// TIA Portal project "ASSEMBLER_3_0" (V18)

(* hardware
DEVICE "S7-1200-Station_1"  S7-1200 Station
   slot 0: "Baugruppenträger_0"  Rack  V1.0
   slot 1: "PLC_2"  CPU 1212C DC/DC/DC  6ES7 212-1AE40-0XB0  V4.6
*)

// ===== PLC "PLC_2"  CPU 1212C DC/DC/DC =====

VAR_GLOBAL   // PLC tag table "Standard-Variablentabelle"
   "System_Byte" AT %MB10 : Byte;
   "FirstScan" AT %M10.0 : Bool;
   "DiagStatusUpdate" AT %M10.1 : Bool;
   "AlwaysTRUE" AT %M10.2 : Bool;
   "AlwaysFALSE" AT %M10.3 : Bool;
   "Clock_Byte" AT %MB20 : Byte;
   "Clock_10Hz" AT %M20.0 : Bool;
   "Clock_5Hz" AT %M20.1 : Bool;
   "Clock_2.5Hz" AT %M20.2 : Bool;
   "Clock_2Hz" AT %M20.3 : Bool;
   "Clock_1.25Hz" AT %M20.4 : Bool;
   "Clock_1Hz" AT %M20.5 : Bool;
   "Clock_0.625Hz" AT %M20.6 : Bool;
   "Clock_0.5Hz" AT %M20.7 : Bool;
   "PART_LEAVING_FE_MEM" AT %M0.2 : Bool;
   "COUNTER_SENSOR_FE_MEM" AT %M0.3 : Bool;
END_VAR

VAR_GLOBAL   // PLC tag table "Tag table from XML_1"
   "LID_AT_PLACE" AT %I0.1 : Bool;
   "BASE_AT_PLACE" AT %I0.2 : Bool;
   "PART_LEAVING" AT %I0.3 : Bool;
   "START_BUTTON" AT %I0.4 : Bool;
   "RESET_BUTTON" AT %I0.5 : Bool;
   "STOP_BUTTON" AT %I0.6 : Bool;
   "EMERGENCY_STOP_BUTTON" AT %I0.7 : Bool;
   "AUTO_SELECTOR" AT %I1.0 : Bool;
   "FACTORY I/O (Running)" AT %I1.1 : Bool;
   "LIDS_CONVEYOR_1" AT %Q0.0 : Bool;
   "STOP_BLADE_1" AT %Q0.1 : Bool;
   "LIDS_CONVEYOR_2" AT %Q0.2 : Bool;
   "BASES_CONVEYOR_1" AT %Q0.3 : Bool;
   "STOP_BLADE_2" AT %Q0.4 : Bool;
   "BASES_CONVEYOR_2" AT %Q0.5 : Bool;
   "GRAB" AT %Q0.6 : Bool;
   "GREEN_LIGHT" AT %Q0.7 : Bool;
   "EMERGENCY_LIGHT" AT %Q1.0 : Bool;
   "RED_LIGHT" AT %Q1.1 : Bool;
   "X" AT %ID30 : Real;
   "Z" AT %ID34 : Real;
   "SET_X" AT %QD30 : Real;
   "SET_Z" AT %QD34 : Real;
   "COUNTER" AT %QD38 : DInt;
   "VAL_BUTTON" AT %I1.4 : Bool;
   "MANUAL_SELECTOR" AT %I1.3 : Bool;
   "ITEM_DETECTED" AT %I0.0 : Bool;
   "STOP_REQUEST" AT %M0.0 : Bool;
   "IN_PRODUCTION" AT %M0.1 : Bool;
   "YELLOW_LIGHT" AT %Q1.2 : Bool;
   "COUNT_SENSOR" AT %I1.2 : Bool;
END_VAR

DATA_BLOCK "DB"   // DB1
{ S7_Optimized_Access := 'TRUE' }
VERSION : 0.1
   VAR
      MODE_REPOS : Bool;
      MODE_MANUEL : Bool;
      MODE_AUTO : Bool;
      MODE_ARU : Bool;
   END_VAR
BEGIN
END_DATA_BLOCK

DATA_BLOCK "FB_AUTO_DB"   // DB5
{ S7_Optimized_Access := 'TRUE' }
VERSION : 0.1
// stored: InstanceOfName FB_AUTO
"FB_AUTO"
BEGIN
END_DATA_BLOCK

DATA_BLOCK "FB_MAN_DB"   // DB6
{ S7_Optimized_Access := 'TRUE' }
VERSION : 0.1
// stored: InstanceOfName FB_MAN
"FB_MAN"
BEGIN
END_DATA_BLOCK

// folder: System blocks/Program resources

DATA_BLOCK "IEC_Counter_0_DB"   // DB2
{ S7_Optimized_Access := 'TRUE' }
AUTHOR : Simatic
FAMILY : IEC
NAME : CNTR
VERSION : 1.0
// stored: InstanceOfName IEC_COUNTER
"IEC_COUNTER"
BEGIN
END_DATA_BLOCK

DATA_BLOCK "IEC_Timer_0_DB_2"   // DB3
{ S7_Optimized_Access := 'TRUE' }
AUTHOR : Simatic
FAMILY : IEC
NAME : IEC_TMR
VERSION : 1.0
// stored: InstanceOfName IEC_TIMER
"IEC_TIMER"
BEGIN
END_DATA_BLOCK

DATA_BLOCK "IEC_Timer_0_DB"   // DB4
{ S7_Optimized_Access := 'TRUE' }
AUTHOR : Simatic
FAMILY : IEC
NAME : IEC_TMR
VERSION : 1.0
// stored: InstanceOfName IEC_TIMER
"IEC_TIMER"
BEGIN
END_DATA_BLOCK

// folder: (top level)

FUNCTION_BLOCK "FB_AUTO"   // FB1, LAD
{ S7_Optimized_Access := 'TRUE' }
VERSION : 0.1
   VAR_INPUT
      part_leaving : Bool;
      Item_detected : Bool;
      lid_at_place : Bool;
      base_at_place : Bool;
      start_button : Bool;
   END_VAR
   VAR_OUTPUT
      lids_conveyor_1 : Bool;
      lids_conveyor_2 : Bool;
      stop_blade_1 : Bool;
      bases_conveyor_1 : Bool;
      bases_coveyor_2 : Bool;
      stop_blade_2 : Bool;
      set_x : Real;
      set_z : Real;
   END_VAR
   VAR_IN_OUT
      grab : Bool;
      in_production : Bool;
   END_VAR
   VAR
      brake : Bool;
      assembled : Bool;
      bases_stop_blade_timer : Bool;
      SR_1 : Bool;
      SR_2 : Bool;
      SR_3 : Bool;
      grab_negative : Bool;
      falling_edge_1 : Bool;
      falling_edge_2 : Bool;
   END_VAR
   VAR_TEMP   // added for the SCL form of the ladder/FBD networks
      _w1 : Bool;
      _w2 : Bool;
   END_VAR
BEGIN

REGION Network 1
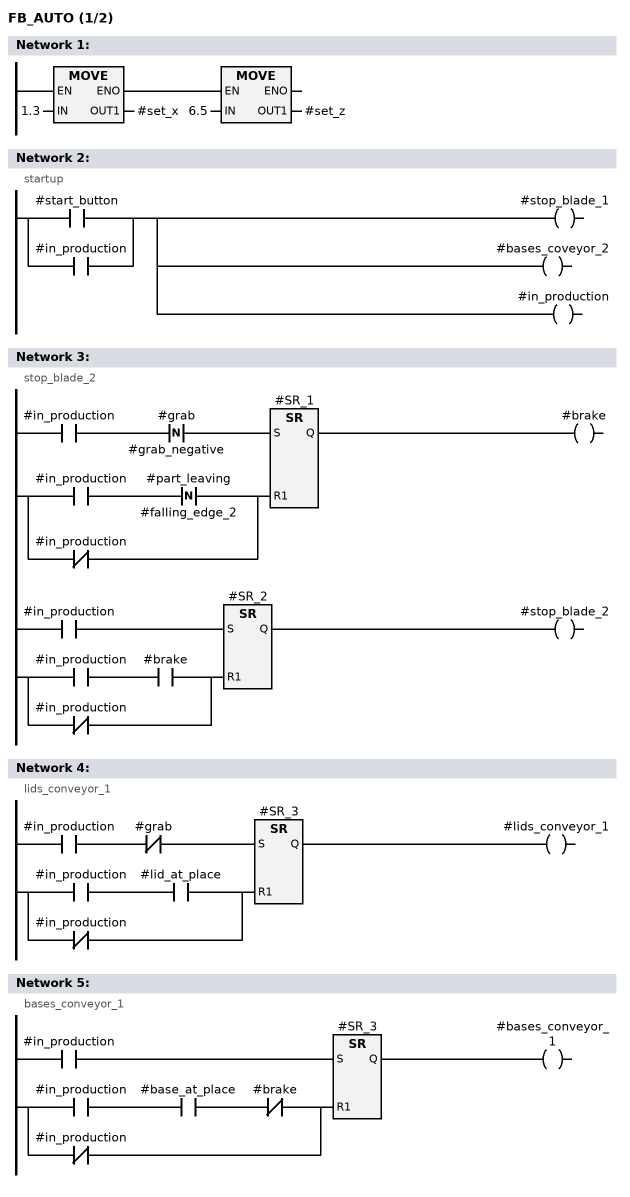
   RUNG wire#powerrail
      Move(in := 1.3, out1 => #set_x)
      Move(in := 6.5, out1 => #set_z)
   END_RUNG
   // the same network as SCL:
   #set_x := 1.3;
   #set_z := 6.5;
END_REGION

REGION Network 2
   // startup
   RUNG wire#powerrail
      Contact( #start_button )
      wire#w1
      Coil( #stop_blade_1 )
   END_RUNG
   RUNG wire#powerrail
      Contact( #in_production )
   END_RUNG wire#w1
   RUNG wire#w1
      Coil( #bases_coveyor_2 )
   END_RUNG
   RUNG wire#w1
      Coil( #in_production )
   END_RUNG
   // the same network as SCL:
   #stop_blade_1 := #start_button OR #in_production;
   #bases_coveyor_2 := #stop_blade_1;
   #in_production := #stop_blade_1;
END_REGION

REGION Network 3
   // stop_blade_2
   RUNG wire#powerrail
      Contact( #in_production )
      N_Contact(operand := #grab, bit := #grab_negative)
      S_SR(operand := #SR_1, r1 := wire#w1)
      Coil( #brake )
   END_RUNG
   RUNG wire#powerrail
      Contact( #in_production )
      N_Contact(operand := #part_leaving, bit := #falling_edge_2)
   END_RUNG wire#w1
   RUNG wire#powerrail
      I_Contact( #in_production )
   END_RUNG wire#w1
   RUNG wire#powerrail
      Contact( #in_production )
      S_SR(operand := #SR_2, r1 := wire#w2)
      Coil( #stop_blade_2 )
   END_RUNG
   RUNG wire#powerrail
      Contact( #in_production )
      Contact( #brake )
   END_RUNG wire#w2
   RUNG wire#powerrail
      I_Contact( #in_production )
   END_RUNG wire#w2
   // the same network as SCL:
   #_w1 := #in_production AND NOT #grab AND #grab_negative;   // falling edge of #grab
   #grab_negative := #grab;
   #_w2 := #in_production AND NOT #part_leaving AND #falling_edge_2;   // falling edge of #part_leaving
   #falling_edge_2 := #part_leaving;
   IF #_w1 THEN
       #SR_1 := TRUE;   // SR flip-flop
   END_IF;
   IF #_w2 OR NOT #in_production THEN #SR_1 := FALSE; END_IF;
   #brake := #SR_1;
   IF #in_production THEN
       #SR_2 := TRUE;   // SR flip-flop
   END_IF;
   IF (#in_production AND #brake) OR NOT #in_production THEN #SR_2 := FALSE; END_IF;
   #stop_blade_2 := #SR_2;
END_REGION

REGION Network 4
   // lids_conveyor_1
   RUNG wire#powerrail
      Contact( #in_production )
      I_Contact( #grab )
      S_SR(operand := #SR_3, r1 := wire#w1)
      Coil( #lids_conveyor_1 )
   END_RUNG
   RUNG wire#powerrail
      Contact( #in_production )
      Contact( #lid_at_place )
   END_RUNG wire#w1
   RUNG wire#powerrail
      I_Contact( #in_production )
   END_RUNG wire#w1
   // the same network as SCL:
   IF #in_production AND NOT #grab THEN
       #SR_3 := TRUE;   // SR flip-flop
   END_IF;
   IF (#in_production AND #lid_at_place) OR NOT #in_production THEN #SR_3 := FALSE; END_IF;
   #lids_conveyor_1 := #SR_3;
END_REGION

REGION Network 5
   // bases_conveyor_1
   RUNG wire#powerrail
      Contact( #in_production )
      S_SR(operand := #SR_3, r1 := wire#w1)
      Coil( #bases_conveyor_1 )
   END_RUNG
   RUNG wire#powerrail
      Contact( #in_production )
      Contact( #base_at_place )
      I_Contact( #brake )
   END_RUNG wire#w1
   RUNG wire#powerrail
      I_Contact( #in_production )
   END_RUNG wire#w1
   // the same network as SCL:
   IF #in_production THEN
       #SR_3 := TRUE;   // SR flip-flop
   END_IF;
   IF (#in_production AND #base_at_place AND NOT #brake) OR NOT #in_production THEN #SR_3 := FALSE; END_IF;
   #bases_conveyor_1 := #SR_3;
END_REGION

REGION Network 6
   // control_de_bras_robotique
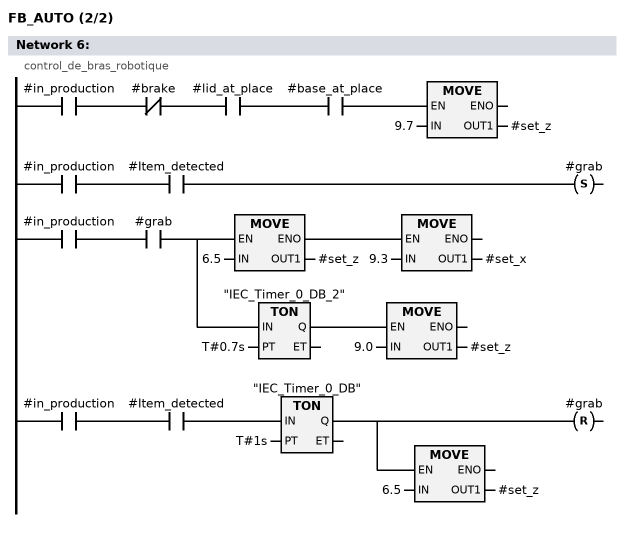
   IF #in_production AND NOT #brake AND #lid_at_place AND #base_at_place THEN #set_z := 9.7; END_IF;
   IF #in_production AND #Item_detected THEN #grab := TRUE; END_IF;
   #_w1 := #in_production AND #grab;
   IF #_w1 THEN
       #set_z := 6.5;
       #set_x := 9.3;
   END_IF;
   "IEC_Timer_0_DB_2".TON(IN := #_w1, PT := T#0.7s);
   IF "IEC_Timer_0_DB_2".Q THEN #set_z := 9.0; END_IF;
   "IEC_Timer_0_DB".TON(IN := #in_production AND #Item_detected, PT := T#1s);
   IF "IEC_Timer_0_DB".Q THEN
       #grab := FALSE;
       #set_z := 6.5;
   END_IF;
END_REGION
END_FUNCTION_BLOCK

FUNCTION_BLOCK "FB_MAN"   // FB2, LAD
{ S7_Optimized_Access := 'TRUE' }
VERSION : 0.1
   VAR_INPUT
      part_leaving : Bool;
      Item_detected : Bool;
      lid_at_place : Bool;
      base_at_place : Bool;
      start_button : Bool;
   END_VAR
   VAR_OUTPUT
      lids_conveyor_1 : Bool;
      lids_conveyor_2 : Bool;
      stop_blade_1 : Bool;
      bases_conveyor_1 : Bool;
      bases_coveyor_2 : Bool;
      stop_blade_2 : Bool;
      set_x : Real;
      set_z : Real;
   END_VAR
   VAR_IN_OUT
      grab : Bool;
      in_production : Bool;
   END_VAR
   VAR
      brake : Bool;
      assembled : Bool;
      bases_stop_blade_timer : Bool;
      SR_1 : Bool;
      SR_2 : Bool;
      SR_3 : Bool;
      grab_negative : Bool;
      falling_edge_1 : Bool;
      falling_edge_2 : Bool;
   END_VAR
   VAR_TEMP   // added for the SCL form of the ladder/FBD networks
      _w1 : Bool;
      _w2 : Bool;
   END_VAR
BEGIN

REGION Network 1
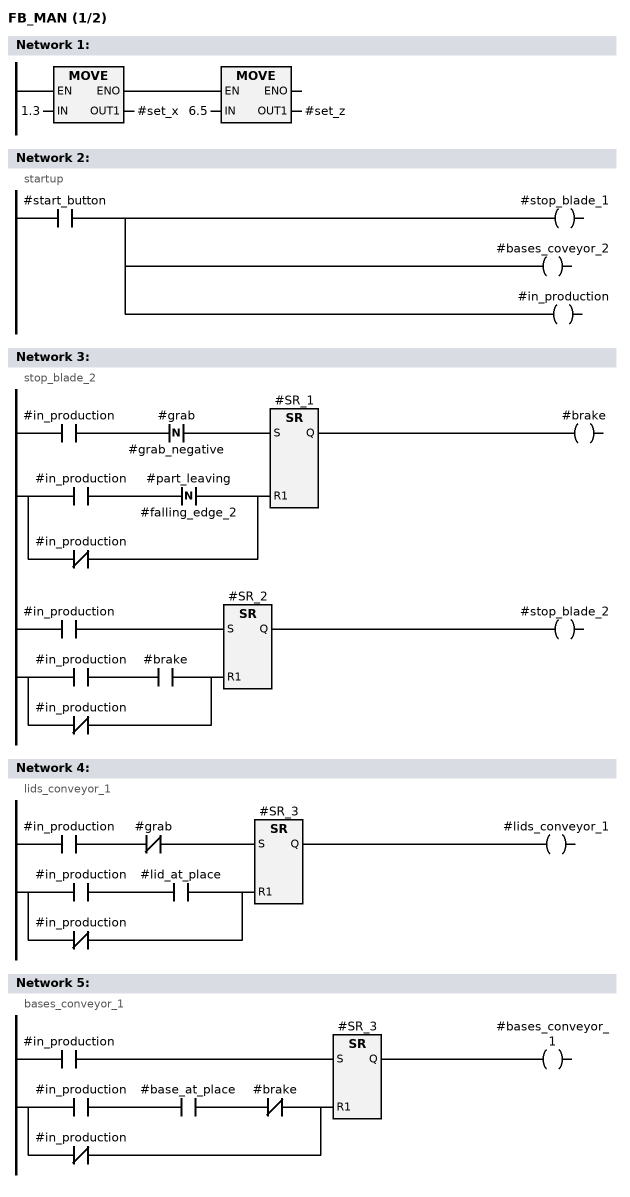
   RUNG wire#powerrail
      Move(in := 1.3, out1 => #set_x)
      Move(in := 6.5, out1 => #set_z)
   END_RUNG
   // the same network as SCL:
   #set_x := 1.3;
   #set_z := 6.5;
END_REGION

REGION Network 2
   // startup
   RUNG wire#powerrail
      Contact( #start_button )
      wire#w1
      Coil( #stop_blade_1 )
   END_RUNG
   RUNG wire#w1
      Coil( #bases_coveyor_2 )
   END_RUNG
   RUNG wire#w1
      Coil( #in_production )
   END_RUNG
   // the same network as SCL:
   #stop_blade_1 := #start_button;
   #bases_coveyor_2 := #start_button;
   #in_production := #start_button;
END_REGION

REGION Network 3
   // stop_blade_2
   RUNG wire#powerrail
      Contact( #in_production )
      N_Contact(operand := #grab, bit := #grab_negative)
      S_SR(operand := #SR_1, r1 := wire#w1)
      Coil( #brake )
   END_RUNG
   RUNG wire#powerrail
      Contact( #in_production )
      N_Contact(operand := #part_leaving, bit := #falling_edge_2)
   END_RUNG wire#w1
   RUNG wire#powerrail
      I_Contact( #in_production )
   END_RUNG wire#w1
   RUNG wire#powerrail
      Contact( #in_production )
      S_SR(operand := #SR_2, r1 := wire#w2)
      Coil( #stop_blade_2 )
   END_RUNG
   RUNG wire#powerrail
      Contact( #in_production )
      Contact( #brake )
   END_RUNG wire#w2
   RUNG wire#powerrail
      I_Contact( #in_production )
   END_RUNG wire#w2
   // the same network as SCL:
   #_w1 := #in_production AND NOT #grab AND #grab_negative;   // falling edge of #grab
   #grab_negative := #grab;
   #_w2 := #in_production AND NOT #part_leaving AND #falling_edge_2;   // falling edge of #part_leaving
   #falling_edge_2 := #part_leaving;
   IF #_w1 THEN
       #SR_1 := TRUE;   // SR flip-flop
   END_IF;
   IF #_w2 OR NOT #in_production THEN #SR_1 := FALSE; END_IF;
   #brake := #SR_1;
   IF #in_production THEN
       #SR_2 := TRUE;   // SR flip-flop
   END_IF;
   IF (#in_production AND #brake) OR NOT #in_production THEN #SR_2 := FALSE; END_IF;
   #stop_blade_2 := #SR_2;
END_REGION

REGION Network 4
   // lids_conveyor_1
   RUNG wire#powerrail
      Contact( #in_production )
      I_Contact( #grab )
      S_SR(operand := #SR_3, r1 := wire#w1)
      Coil( #lids_conveyor_1 )
   END_RUNG
   RUNG wire#powerrail
      Contact( #in_production )
      Contact( #lid_at_place )
   END_RUNG wire#w1
   RUNG wire#powerrail
      I_Contact( #in_production )
   END_RUNG wire#w1
   // the same network as SCL:
   IF #in_production AND NOT #grab THEN
       #SR_3 := TRUE;   // SR flip-flop
   END_IF;
   IF (#in_production AND #lid_at_place) OR NOT #in_production THEN #SR_3 := FALSE; END_IF;
   #lids_conveyor_1 := #SR_3;
END_REGION

REGION Network 5
   // bases_conveyor_1
   RUNG wire#powerrail
      Contact( #in_production )
      S_SR(operand := #SR_3, r1 := wire#w1)
      Coil( #bases_conveyor_1 )
   END_RUNG
   RUNG wire#powerrail
      Contact( #in_production )
      Contact( #base_at_place )
      I_Contact( #brake )
   END_RUNG wire#w1
   RUNG wire#powerrail
      I_Contact( #in_production )
   END_RUNG wire#w1
   // the same network as SCL:
   IF #in_production THEN
       #SR_3 := TRUE;   // SR flip-flop
   END_IF;
   IF (#in_production AND #base_at_place AND NOT #brake) OR NOT #in_production THEN #SR_3 := FALSE; END_IF;
   #bases_conveyor_1 := #SR_3;
END_REGION

REGION Network 6
   // control_de_bras_robotique
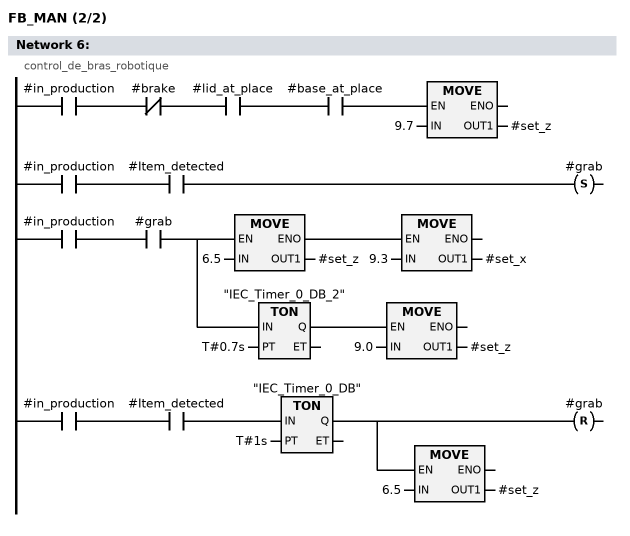
   IF #in_production AND NOT #brake AND #lid_at_place AND #base_at_place THEN #set_z := 9.7; END_IF;
   IF #in_production AND #Item_detected THEN #grab := TRUE; END_IF;
   #_w1 := #in_production AND #grab;
   IF #_w1 THEN
       #set_z := 6.5;
       #set_x := 9.3;
   END_IF;
   "IEC_Timer_0_DB_2".TON(IN := #_w1, PT := T#0.7s);
   IF "IEC_Timer_0_DB_2".Q THEN #set_z := 9.0; END_IF;
   "IEC_Timer_0_DB".TON(IN := #in_production AND #Item_detected, PT := T#1s);
   IF "IEC_Timer_0_DB".Q THEN
       #grab := FALSE;
       #set_z := 6.5;
   END_IF;
END_REGION
END_FUNCTION_BLOCK

FUNCTION "FC_ARU_REPOS" : Void   // FC2, LAD
{ S7_Optimized_Access := 'TRUE' }
VERSION : 0.1
   VAR_OUTPUT
      lids_conveyor_1 : Bool;
      lids_conveyor_2 : Bool;
      stop_blade_1 : Bool;
      bases_conveyor_1 : Bool;
      bases_coveyor_2 : Bool;
      stop_blade_2 : Bool;
   END_VAR
   VAR_IN_OUT
      grab : Bool;
   END_VAR
BEGIN

REGION Network 1
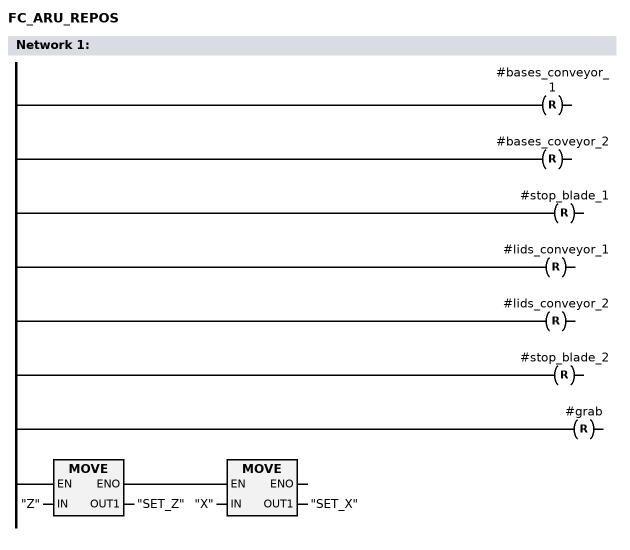
   RUNG wire#powerrail
      R_Coil( #bases_conveyor_1 )
   END_RUNG
   RUNG wire#powerrail
      R_Coil( #bases_coveyor_2 )
   END_RUNG
   RUNG wire#powerrail
      R_Coil( #stop_blade_1 )
   END_RUNG
   RUNG wire#powerrail
      R_Coil( #lids_conveyor_1 )
   END_RUNG
   RUNG wire#powerrail
      R_Coil( #lids_conveyor_2 )
   END_RUNG
   RUNG wire#powerrail
      R_Coil( #stop_blade_2 )
   END_RUNG
   RUNG wire#powerrail
      R_Coil( #grab )
   END_RUNG
   RUNG wire#powerrail
      Move(in := "Z", out1 => "SET_Z")
      Move(in := "X", out1 => "SET_X")
   END_RUNG
   // the same network as SCL:
   #bases_conveyor_1 := FALSE;
   #bases_coveyor_2 := FALSE;
   #stop_blade_1 := FALSE;
   #lids_conveyor_1 := FALSE;
   #lids_conveyor_2 := FALSE;
   #stop_blade_2 := FALSE;
   #grab := FALSE;
   "SET_Z" := "Z";
   "SET_X" := "X";
END_REGION
END_FUNCTION

FUNCTION "FC_MODES_GEST" : Void   // FC5, LAD
{ S7_Optimized_Access := 'TRUE' }
VERSION : 0.1
   VAR_INPUT
      stop_button : Bool;
      auto_selector : Bool;
      val_button : Bool;
      manual_selector : Bool;
      emergency_stop_button : Bool;
      part_leaving : Bool;
   END_VAR
   VAR_OUTPUT
      green_light : Bool;
      yellow_light : Bool;
      red_light : Bool;
      emergency_light : Bool;
   END_VAR
   VAR_IN_OUT
      mode_man : Bool;
      mode_repos : Bool;
      mode_auto : Bool;
      mode_aru : Bool;
      in_production : Bool;
   END_VAR
   VAR_TEMP   // added for the SCL form of the ladder/FBD networks
      _w1 : Bool;
      _w2 : Bool;
   END_VAR
BEGIN

REGION Network 1
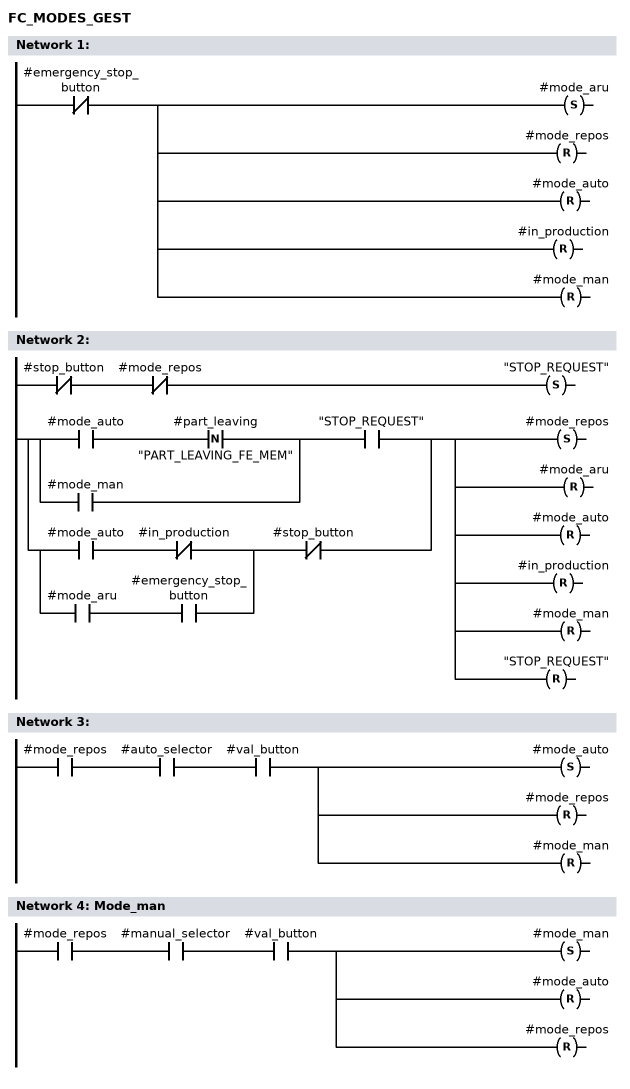
   RUNG wire#powerrail
      I_Contact( #emergency_stop_button )
      wire#w1
      S_Coil( #mode_aru )
   END_RUNG
   RUNG wire#w1
      R_Coil( #mode_repos )
   END_RUNG
   RUNG wire#w1
      R_Coil( #mode_auto )
   END_RUNG
   RUNG wire#w1
      R_Coil( #in_production )
   END_RUNG
   RUNG wire#w1
      R_Coil( #mode_man )
   END_RUNG
   // the same network as SCL:
   IF NOT #emergency_stop_button THEN
       #mode_aru := TRUE;
       #mode_repos := FALSE;
       #mode_auto := FALSE;
       #in_production := FALSE;
       #mode_man := FALSE;
   END_IF;
END_REGION

REGION Network 2
   RUNG wire#powerrail
      I_Contact( #stop_button )
      I_Contact( #mode_repos )
      S_Coil( "STOP_REQUEST" )
   END_RUNG
   RUNG wire#powerrail
      Contact( #mode_auto )
      N_Contact(operand := #part_leaving, bit := "PART_LEAVING_FE_MEM")
      wire#w1
      Contact( "STOP_REQUEST" )
      wire#w2
      S_Coil( #mode_repos )
   END_RUNG
   RUNG wire#powerrail
      Contact( #mode_man )
   END_RUNG wire#w1
   RUNG wire#powerrail
      Contact( #mode_auto )
      I_Contact( #in_production )
      wire#w3
      I_Contact( #stop_button )
   END_RUNG wire#w2
   RUNG wire#powerrail
      Contact( #mode_aru )
      Contact( #emergency_stop_button )
   END_RUNG wire#w3
   RUNG wire#w2
      R_Coil( #mode_aru )
   END_RUNG
   RUNG wire#w2
      R_Coil( #mode_auto )
   END_RUNG
   RUNG wire#w2
      R_Coil( #in_production )
   END_RUNG
   RUNG wire#w2
      R_Coil( #mode_man )
   END_RUNG
   RUNG wire#w2
      R_Coil( "STOP_REQUEST" )
   END_RUNG
   // the same network as SCL:
   IF NOT #stop_button AND NOT #mode_repos THEN "STOP_REQUEST" := TRUE; END_IF;
   #_w1 := #mode_auto AND NOT #part_leaving AND "PART_LEAVING_FE_MEM";   // falling edge of #part_leaving
   "PART_LEAVING_FE_MEM" := #part_leaving;
   IF ((#_w1 OR #mode_man) AND "STOP_REQUEST") OR (((#mode_auto AND NOT #in_production) OR (#mode_aru AND #emergency_stop_button)) AND NOT #stop_button) THEN
       #mode_repos := TRUE;
   END_IF;
   #_w2 := ((#_w1 OR #mode_man) AND "STOP_REQUEST") OR (((#mode_auto AND NOT #in_production) OR (#mode_aru AND #emergency_stop_button)) AND NOT #stop_button);
   IF #_w2 THEN
       #mode_aru := FALSE;
       #mode_auto := FALSE;
       #in_production := FALSE;
       #mode_man := FALSE;
       "STOP_REQUEST" := FALSE;
   END_IF;
END_REGION

REGION Network 3
   RUNG wire#powerrail
      Contact( #mode_repos )
      Contact( #auto_selector )
      Contact( #val_button )
      wire#w1
      S_Coil( #mode_auto )
   END_RUNG
   RUNG wire#w1
      R_Coil( #mode_repos )
   END_RUNG
   RUNG wire#w1
      R_Coil( #mode_man )
   END_RUNG
   // the same network as SCL:
   IF #mode_repos AND #auto_selector AND #val_button THEN #mode_auto := TRUE; END_IF;
   #_w1 := #mode_repos AND #auto_selector AND #val_button;
   IF #_w1 THEN
       #mode_repos := FALSE;
       #mode_man := FALSE;
   END_IF;
END_REGION

REGION Network 4: Mode_man
   RUNG wire#powerrail
      Contact( #mode_repos )
      Contact( #manual_selector )
      Contact( #val_button )
      wire#w1
      S_Coil( #mode_man )
   END_RUNG
   RUNG wire#w1
      R_Coil( #mode_auto )
   END_RUNG
   RUNG wire#w1
      R_Coil( #mode_repos )
   END_RUNG
   // the same network as SCL:
   IF #mode_repos AND #manual_selector AND #val_button THEN
       #mode_man := TRUE;
       #mode_auto := FALSE;
       #mode_repos := FALSE;
   END_IF;
END_REGION
END_FUNCTION

FUNCTION "FC_VOY_GEST" : Void   // FC6, LAD
{ S7_Optimized_Access := 'TRUE' }
VERSION : 0.1
   VAR_OUTPUT
      green_light : Bool;
      yellow_light : Bool;
      red_light : Bool;
      emergency_light : Bool;
   END_VAR
   VAR_IN_OUT
      mode_man : Bool;
      mode_repos : Bool;
      mode_auto : Bool;
      mode_aru : Bool;
      in_production : Bool;
   END_VAR
BEGIN

REGION Network 1
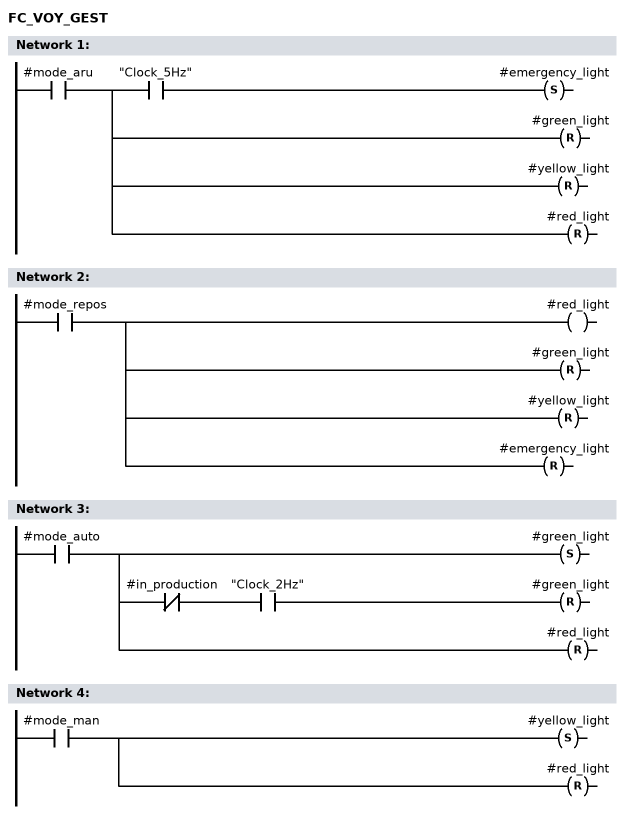
   RUNG wire#powerrail
      Contact( #mode_aru )
      wire#w1
      Contact( "Clock_5Hz" )
      S_Coil( #emergency_light )
   END_RUNG
   RUNG wire#w1
      R_Coil( #green_light )
   END_RUNG
   RUNG wire#w1
      R_Coil( #yellow_light )
   END_RUNG
   RUNG wire#w1
      R_Coil( #red_light )
   END_RUNG
   // the same network as SCL:
   IF #mode_aru AND "Clock_5Hz" THEN #emergency_light := TRUE; END_IF;
   IF #mode_aru THEN
       #green_light := FALSE;
       #yellow_light := FALSE;
       #red_light := FALSE;
   END_IF;
END_REGION

REGION Network 2
   RUNG wire#powerrail
      Contact( #mode_repos )
      wire#w1
      Coil( #red_light )
   END_RUNG
   RUNG wire#w1
      R_Coil( #green_light )
   END_RUNG
   RUNG wire#w1
      R_Coil( #yellow_light )
   END_RUNG
   RUNG wire#w1
      R_Coil( #emergency_light )
   END_RUNG
   // the same network as SCL:
   #red_light := #mode_repos;
   IF #mode_repos THEN
       #green_light := FALSE;
       #yellow_light := FALSE;
       #emergency_light := FALSE;
   END_IF;
END_REGION

REGION Network 3
   RUNG wire#powerrail
      Contact( #mode_auto )
      wire#w1
      S_Coil( #green_light )
   END_RUNG
   RUNG wire#w1
      I_Contact( #in_production )
      Contact( "Clock_2Hz" )
      R_Coil( #green_light )
   END_RUNG
   RUNG wire#w1
      R_Coil( #red_light )
   END_RUNG
   // the same network as SCL:
   IF #mode_auto THEN #green_light := TRUE; END_IF;
   IF #mode_auto AND NOT #in_production AND "Clock_2Hz" THEN #green_light := FALSE; END_IF;
   IF #mode_auto THEN #red_light := FALSE; END_IF;
END_REGION

REGION Network 4
   RUNG wire#powerrail
      Contact( #mode_man )
      wire#w1
      S_Coil( #yellow_light )
   END_RUNG
   RUNG wire#w1
      R_Coil( #red_light )
   END_RUNG
   // the same network as SCL:
   IF #mode_man THEN
       #yellow_light := TRUE;
       #red_light := FALSE;
   END_IF;
END_REGION

REGION Network 6: Mode_man
END_REGION
END_FUNCTION

FUNCTION "Factory_IO" : Void   // FC9000, SCL
{ S7_Optimized_Access := 'TRUE' }
VERSION : 0.1
   VAR_TEMP
      rdTimeReturn : Int;
      outputTime : DTL;
      SyncVal : Byte;
      forVal : Int;
      forVal_2 : Int;
      Value : Byte;
   END_VAR
   VAR CONSTANT
      CompVal : Byte := 16#34;
      Value_01 : Byte := 16#11;
      Value_01_DW : DWord := 16#A165_D992;
      Value_02_DW : DWord := 16#58BE_4401;
   END_VAR
BEGIN

   #Value:=PEEK(area := 16#82,
        dbNumber := 0,
        byteOffset := 511);
   #Value := #Value + 1;

   POKE(area := 16#82,
        dbNumber := 0,
        byteOffset := 511,
        value := #Value);

   POKE(area:=16#81,
        dbNumber:=0,
        byteOffset:=1016,
        value:=#Value_01_DW);
   POKE(area := 16#81,
        dbNumber := 0,
        byteOffset := 1020,
        value := #Value_02_DW);

   POKE(area := 16#81,
        dbNumber := 0,
        byteOffset := 511,
        value := B#16#00);

   FOR #forVal := 0 TO 120 DO
       FOR #forVal_2:=0 TO 10 DO
           #rdTimeReturn:=RD_SYS_T(#outputTime);
           #rdTimeReturn := WR_SYS_T(#outputTime);
           #rdTimeReturn := RD_SYS_T(#outputTime);
           #rdTimeReturn := WR_SYS_T(#outputTime);
       END_FOR;
       #SyncVal:= PEEK(area := 16#81,
                      dbNumber := 0,
                      byteOffset := 511);
       IF #SyncVal = #CompVal THEN
          GOTO M_1;
       END_IF;
   END_FOR;
   RETURN;

   M_1:
   POKE(area := 16#81,
        dbNumber := 0,
        byteOffset := 511,
        value := B#16#0);
END_FUNCTION

ORGANIZATION_BLOCK "Main"   // OB1, LAD, ProgramCycle
TITLE = "Main Program Sweep (Cycle)"
{ S7_Optimized_Access := 'TRUE' }
VERSION : 0.1
   VAR_INPUT
      Initial_Call : Bool;   // Initial call of this OB
      Remanence : Bool;   // =True, if remanent data are available
   END_VAR
   VAR_TEMP   // added for the SCL form of the ladder/FBD networks
      _w1 : Bool;
   END_VAR
BEGIN

REGION Network 1: Konnektierungsbaustein für PLC-Lab
   // Im Netzwerk 1 wird der Konnektierungsbaustein für PLC-Lab aufgerufen.
   // Dieser Aufruf darf nicht entfernt werden!
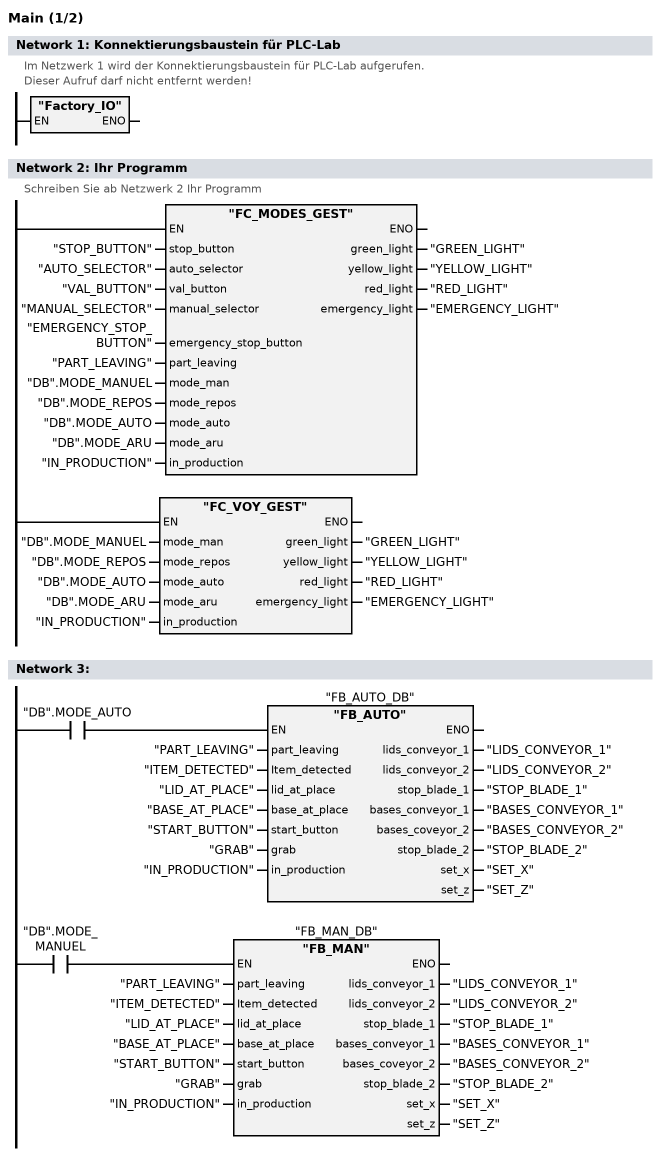
   RUNG wire#powerrail
      "Factory_IO"()
   END_RUNG
   // the same network as SCL:
   "Factory_IO"();
END_REGION

REGION Network 2: Ihr Programm
   // Schreiben Sie ab Netzwerk 2 Ihr Programm
   RUNG wire#powerrail
      "FC_MODES_GEST"(stop_button := "STOP_BUTTON", auto_selector := "AUTO_SELECTOR", val_button := "VAL_BUTTON", manual_selector := "MANUAL_SELECTOR", emergency_stop_button := "EMERGENCY_STOP_BUTTON", part_leaving := "PART_LEAVING", mode_man := "DB".MODE_MANUEL, mode_repos := "DB".MODE_REPOS, mode_auto := "DB".MODE_AUTO, mode_aru := "DB".MODE_ARU, in_production := "IN_PRODUCTION", green_light => "GREEN_LIGHT", yellow_light => "YELLOW_LIGHT", red_light => "RED_LIGHT", emergency_light => "EMERGENCY_LIGHT")
   END_RUNG
   RUNG wire#powerrail
      "FC_VOY_GEST"(mode_man := "DB".MODE_MANUEL, mode_repos := "DB".MODE_REPOS, mode_auto := "DB".MODE_AUTO, mode_aru := "DB".MODE_ARU, in_production := "IN_PRODUCTION", green_light => "GREEN_LIGHT", yellow_light => "YELLOW_LIGHT", red_light => "RED_LIGHT", emergency_light => "EMERGENCY_LIGHT")
   END_RUNG
   // the same network as SCL:
   "FC_MODES_GEST"(stop_button := "STOP_BUTTON",
                   auto_selector := "AUTO_SELECTOR",
                   val_button := "VAL_BUTTON",
                   manual_selector := "MANUAL_SELECTOR",
                   emergency_stop_button := "EMERGENCY_STOP_BUTTON",
                   part_leaving := "PART_LEAVING",
                   mode_man := "DB".MODE_MANUEL,
                   mode_repos := "DB".MODE_REPOS,
                   mode_auto := "DB".MODE_AUTO,
                   mode_aru := "DB".MODE_ARU,
                   in_production := "IN_PRODUCTION",
                   green_light => "GREEN_LIGHT",
                   yellow_light => "YELLOW_LIGHT",
                   red_light => "RED_LIGHT",
                   emergency_light => "EMERGENCY_LIGHT");
   "FC_VOY_GEST"(mode_man := "DB".MODE_MANUEL,
                 mode_repos := "DB".MODE_REPOS,
                 mode_auto := "DB".MODE_AUTO,
                 mode_aru := "DB".MODE_ARU,
                 in_production := "IN_PRODUCTION",
                 green_light => "GREEN_LIGHT",
                 yellow_light => "YELLOW_LIGHT",
                 red_light => "RED_LIGHT",
                 emergency_light => "EMERGENCY_LIGHT");
END_REGION

REGION Network 3
   RUNG wire#powerrail
      Contact( "DB".MODE_AUTO )
      "FB_AUTO_DB"(part_leaving := "PART_LEAVING", Item_detected := "ITEM_DETECTED", lid_at_place := "LID_AT_PLACE", base_at_place := "BASE_AT_PLACE", start_button := "START_BUTTON", grab := "GRAB", in_production := "IN_PRODUCTION", lids_conveyor_1 => "LIDS_CONVEYOR_1", lids_conveyor_2 => "LIDS_CONVEYOR_2", stop_blade_1 => "STOP_BLADE_1", bases_conveyor_1 => "BASES_CONVEYOR_1", bases_coveyor_2 => "BASES_CONVEYOR_2", stop_blade_2 => "STOP_BLADE_2", set_x => "SET_X", set_z => "SET_Z")
   END_RUNG
   RUNG wire#powerrail
      Contact( "DB".MODE_MANUEL )
      "FB_MAN_DB"(part_leaving := "PART_LEAVING", Item_detected := "ITEM_DETECTED", lid_at_place := "LID_AT_PLACE", base_at_place := "BASE_AT_PLACE", start_button := "START_BUTTON", grab := "GRAB", in_production := "IN_PRODUCTION", lids_conveyor_1 => "LIDS_CONVEYOR_1", lids_conveyor_2 => "LIDS_CONVEYOR_2", stop_blade_1 => "STOP_BLADE_1", bases_conveyor_1 => "BASES_CONVEYOR_1", bases_coveyor_2 => "BASES_CONVEYOR_2", stop_blade_2 => "STOP_BLADE_2", set_x => "SET_X", set_z => "SET_Z")
   END_RUNG
   // the same network as SCL:
   IF "DB".MODE_AUTO THEN
       "FB_AUTO_DB"(part_leaving := "PART_LEAVING",   // "FB_AUTO"
                    Item_detected := "ITEM_DETECTED",
                    lid_at_place := "LID_AT_PLACE",
                    base_at_place := "BASE_AT_PLACE",
                    start_button := "START_BUTTON",
                    grab := "GRAB",
                    in_production := "IN_PRODUCTION",
                    lids_conveyor_1 => "LIDS_CONVEYOR_1",
                    lids_conveyor_2 => "LIDS_CONVEYOR_2",
                    stop_blade_1 => "STOP_BLADE_1",
                    bases_conveyor_1 => "BASES_CONVEYOR_1",
                    bases_coveyor_2 => "BASES_CONVEYOR_2",
                    stop_blade_2 => "STOP_BLADE_2",
                    set_x => "SET_X",
                    set_z => "SET_Z");
   END_IF;
   IF "DB".MODE_MANUEL THEN
       "FB_MAN_DB"(part_leaving := "PART_LEAVING",   // "FB_MAN"
                   Item_detected := "ITEM_DETECTED",
                   lid_at_place := "LID_AT_PLACE",
                   base_at_place := "BASE_AT_PLACE",
                   start_button := "START_BUTTON",
                   grab := "GRAB",
                   in_production := "IN_PRODUCTION",
                   lids_conveyor_1 => "LIDS_CONVEYOR_1",
                   lids_conveyor_2 => "LIDS_CONVEYOR_2",
                   stop_blade_1 => "STOP_BLADE_1",
                   bases_conveyor_1 => "BASES_CONVEYOR_1",
                   bases_coveyor_2 => "BASES_CONVEYOR_2",
                   stop_blade_2 => "STOP_BLADE_2",
                   set_x => "SET_X",
                   set_z => "SET_Z");
   END_IF;
END_REGION

REGION Network 4
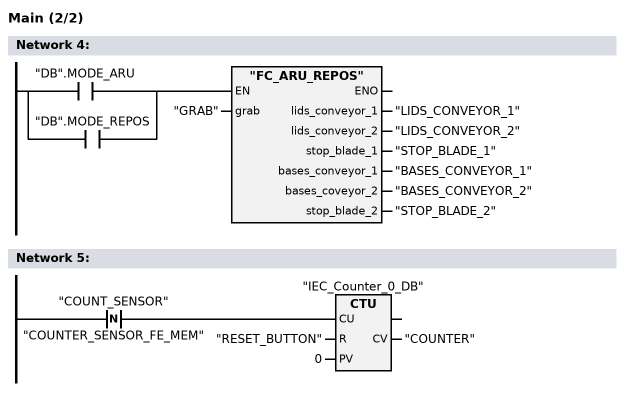
   RUNG wire#powerrail
      Contact( "DB".MODE_ARU )
      wire#w1
      "FC_ARU_REPOS"(grab := "GRAB", lids_conveyor_1 => "LIDS_CONVEYOR_1", lids_conveyor_2 => "LIDS_CONVEYOR_2", stop_blade_1 => "STOP_BLADE_1", bases_conveyor_1 => "BASES_CONVEYOR_1", bases_coveyor_2 => "BASES_CONVEYOR_2", stop_blade_2 => "STOP_BLADE_2")
   END_RUNG
   RUNG wire#powerrail
      Contact( "DB".MODE_REPOS )
   END_RUNG wire#w1
   // the same network as SCL:
   IF "DB".MODE_ARU OR "DB".MODE_REPOS THEN
       "FC_ARU_REPOS"(grab := "GRAB",
                      lids_conveyor_1 => "LIDS_CONVEYOR_1",
                      lids_conveyor_2 => "LIDS_CONVEYOR_2",
                      stop_blade_1 => "STOP_BLADE_1",
                      bases_conveyor_1 => "BASES_CONVEYOR_1",
                      bases_coveyor_2 => "BASES_CONVEYOR_2",
                      stop_blade_2 => "STOP_BLADE_2");
   END_IF;
END_REGION

REGION Network 5
   #_w1 := NOT "COUNT_SENSOR" AND "COUNTER_SENSOR_FE_MEM";   // falling edge of "COUNT_SENSOR"
   "COUNTER_SENSOR_FE_MEM" := "COUNT_SENSOR";
   "IEC_Counter_0_DB".CTU(CU := #_w1, R := "RESET_BUTTON", PV := 0, CV => "COUNTER");
END_REGION
END_ORGANIZATION_BLOCK

ORGANIZATION_BLOCK "Startup"   // OB100, LAD, Startup
TITLE = "Complete Restart"
{ S7_Optimized_Access := 'TRUE' }
VERSION : 0.1
   VAR_INPUT
      LostRetentive : Bool;   // True if retentive data are lost
      LostRTC : Bool;   // True if date and time are lost
   END_VAR
BEGIN

REGION Network 1
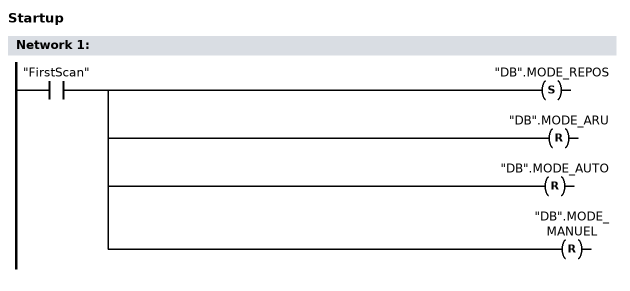
   RUNG wire#powerrail
      Contact( "FirstScan" )
      wire#w1
      S_Coil( "DB".MODE_REPOS )
   END_RUNG
   RUNG wire#w1
      R_Coil( "DB".MODE_ARU )
   END_RUNG
   RUNG wire#w1
      R_Coil( "DB".MODE_AUTO )
   END_RUNG
   RUNG wire#w1
      R_Coil( "DB".MODE_MANUEL )
   END_RUNG
   // the same network as SCL:
   IF "FirstScan" THEN
       "DB".MODE_REPOS := TRUE;
       "DB".MODE_ARU := FALSE;
       "DB".MODE_AUTO := FALSE;
       "DB".MODE_MANUEL := FALSE;
   END_IF;
END_REGION
END_ORGANIZATION_BLOCK